// TIA Portal V18 export
// export: Created 2025-12-01T17:52:52.7143684Z, ExportSetting None, DisplayName Totally Integrated Automation Portal, DisplayVersion V18 Update 5, DisplayName TIA Portal Openness, DisplayVersion V18 Update 5, DisplayName TIA Portal Teamcenter Gateway, DisplayVersion V18, DisplayName TIA Portal Version Control Interface, DisplayVersion V18, DisplayName STEP 7 Professional, DisplayVersion V18 Update 5, DisplayName STEP 7 Safety, DisplayVersion V18, DisplayName WinCC Professional, DisplayVersion V18 Update 5
Screen "10MainScreen"  1280x800, Number=10, Template=00MainScreen
  on GenerateScreen: SetBit(Tag := NormalON); ResetBit(Tag := NormalOFF); SetTag(Tag := ST_SysDBNum, Value := 1060); SetTag(Tag := PM_CountCycleDBNum, Value := 1061); SetTag(Tag := ST_PMDBNum, Value := 1063)
  ScreenLayer "Layer_0"
    Button "按钮_4" at 383,725 size 128x75  PictureOff=向右箭头_0, StyleItem=BtnNormal20, TextOff="报 警 / Alarm / Poplach"
      RangeAppearanceAnimation "RangeAppearanceAnimation"
        tag ST_AlarmON
        1..1: back #ff0000, fore #d6d3ce, flashing
      on Click: ActivateScreen(Screen name := 300Main, Object number := 0); SetTag(Tag := Sys_VersionManagement_HMIPageID, Value := 300)
    Button "按钮_6"  Authorization=Manage Parameter, PictureOff=向右箭头_0, StyleItem=BtnNormal20, TextOff="参数设定 / Parameter setting / Parameter nastavenie", TextOn="参数设定 / Parameter setting / Parameter nastavenie"
      RangeAppearanceAnimation "RangeAppearanceAnimation"
        tag _unlock[5]
        0..0: back #d6e1e8, fore #c0c0c0
      on Click: ActivateScreen(Screen name := 700 Main, Object number := 0)
    Button "按钮_8" at 511,725 size 128x75  StyleItem=BtnNormal20, TextOff="MES", TextOn="照明灯 / Light / Svetlo"
      on Press: ActivateScreen(Screen name := 900MES, Object number := 0); SetTag(Tag := Sys_VersionManagement_HMIPageID, Value := 900)
    Button "按钮_11" at 256,725 size 128x75  PictureOff=向右箭头_0, StyleItem=BtnNormal20, TextOff="Safety Status", TextOn="Safety Status"
      on Click: ShowPopupScreen(Name of the screen := Pilz, X coordinate := 350, Y coordinate := 150, Display mode := -1, Animation := -1, Animation speed := 1)
    Button "btnMenu5_1" at 128,725 size 128x75  StyleItem=BtnActive20, TextOff="主页面 / Main", TextOn="主页面 / Main"
      on Click: ActivateScreen(Screen name := , Object number := 0); SetTag(Tag := Sys_VersionManagement_HMIPageID, Value := 10)
    Button "按钮_1"  PictureOff=向右箭头_0, StyleItem=BtnNormal20, TextList=蜂鸣器屏蔽, TextOff="蜂鸣器 屏蔽 / Buzzer shield / Bzučiak štít", TextOn="蜂鸣器 屏蔽 / Buzzer shield"
      RangeAppearanceAnimation "RangeAppearanceAnimation"
        tag ST_CommandBuzzerOn
        1..1: back #3366ff, fore #d6d3ce
      on Click: InvertBit(Tag := ST_CommandBuzzerOn)
      ProcessValue := ST_CommandBuzzerOn
    GraphicView "图形视图_1" at 157,95 size 972x584  Picture=图形_44
    Circle "圆_1" at 259,725 size 29x29
      RangeAppearanceAnimation "RangeAppearanceAnimation"
        tag PilzData_Status
        1..1: back #00ff00, fore #181c31
        2..2: back #ff0000, fore #181c31
    TextField "文本域_14" at 227,649 size 17x28  Text="1"
    TextField "文本域_9" at 1132,93 size 118x42  Text="Current Temperature_1 / Text"
    TextField "文本域_10" at 1132,130 size 118x42  Text="Current Temperature_2 / Text"
    TextField "文本域_11" at 1132,177 size 125x23  Text="SetTemperature / Text"
    TextField "文本域_12" at 1133,213 size 117x23  Text="SetSolidifyTime / Text"
    TextField "文本域_13" at 1132,241 size 92x42  Text="Actual SolidifyTime / Text"
    IOField "I/O 域_1"  FormatPattern=s99999, Mode=Output, ShiftDecimalPoint=1
      ProcessValue := ST10_PLC_GetDB_InData_Data_CurrentTemperature_1
    IOField "I/O 域_2"  FormatPattern=s99999, Mode=Output, ShiftDecimalPoint=1
      ProcessValue := ST10_PLC_GetDB_InData_Data_CurrentTemperature_2
    IOField "I/O 域_3"  FormatPattern=s99999, Mode=Output, ShiftDecimalPoint=1
      ProcessValue := ST10_PLC_GetDB_InData_Data_SetTemperature
    IOField "I/O 域_4"  FormatPattern=s99999, Mode=Output, Unit=min
      ProcessValue := ST10_PLC_GetDB_InData_Data_SetSolidifyTime
    IOField "I/O 域_5"  FormatPattern=s99999, Mode=Output, Unit=min
      ProcessValue := ST10_PLC_GetDB_InData_Data_ActualSolidifyTime
    SymbolicIOField "符号 IO 域_5" at 291,96 size 742x36  Mode=Output, TextList=FlowName5, TextOff="0", TextOn="1"
      ProcessValue := "ST_PMStep[5]"
    Rectangle "矩形_1" at 1037,283 size 176x159
    Circle "圆_17" at 1047,321 size 17x17
      RangeAppearanceAnimation "RangeAppearanceAnimation"
        tag ST10_PLC_GetDB_InData_Global_Beat
        0..0: back #d9d9d9, fore #181c31
        1..1: back #00ff00, fore #181c31
    TextField "文本域_1" at 1079,316 size 48x28  Text="Beat / Text"
    Circle "圆_18" at 1047,349 size 17x17
      RangeAppearanceAnimation "RangeAppearanceAnimation"
        tag ST10_PLC_GetDB_InData_Global_Alarm
        0..0: back #d9d9d9, fore #181c31
        1..1: back #ff0000, fore #181c31
    TextField "文本域_3"  Text="Alarm / Text"
    Circle "圆_19" at 1047,378 size 17x17
      RangeAppearanceAnimation "RangeAppearanceAnimation"
        tag ST10_PLC_GetDB_InData_Global_AutoMode
        1..1: back #00ff00, fore #181c31
        0..0: back #d9d9d9, fore #181c31
    TextField "文本域_5" at 1079,372 size 101x28  Text="AutoMode / Text"
    Circle "圆_20" at 1047,407 size 17x17
      RangeAppearanceAnimation "RangeAppearanceAnimation"
        tag ST10_PLC_GetDB_InData_Global_ManualMode
        1..1: back #00ff00, fore #181c31
        0..0: back #d9d9d9, fore #181c31
    TextField "文本域_6" at 1079,401 size 124x28  Text="ManualMode / Text"
    TextField "文本域_2" at 1064,286 size 139x28  Text="固化炉 / SolidifyStatus"
    Rectangle "矩形_2" at 172,95 size 117x37
    TextField "文本域_4" at 196,100 size 82x28  Text="ROBOT1"
    SymbolicIOField "符号 IO 域_1" at 291,136 size 742x36  Mode=Output, TextList=FlowName8, TextOff="0", TextOn="1"
      ProcessValue := "ST_PMStep[8]"
    Rectangle "矩形_3" at 172,135 size 117x37
    TextField "文本域_7" at 196,140 size 82x28  Text="ROBOT2"
    SymbolicIOField "符号 IO 域_2" at 291,176 size 742x36  Mode=Output, TextList=FlowName15, TextOff="0", TextOn="1"
      ProcessValue := "ST_PMStep[15]"
    Rectangle "矩形_4" at 172,175 size 117x37
    TextField "文本域_8" at 196,180 size 82x28  Text="ROBOT3"
    IOField "I/O 域_6" at 290,644 size 107x32  FormatPattern=999, Unit=%
      ProcessValue := KukaRobot1_CtrlDB_iSpeedValue
    TextField "文本域_15" at 158,648 size 131x28  Text="Robot1Speed:"
    IOField "I/O 域_7" at 541,644 size 107x32  FormatPattern=999, Unit=%
      ProcessValue := KukaRobot2_CtrlDB_iSpeedValue
    TextField "文本域_16" at 409,648 size 131x28  Text="Robot2Speed:"
    IOField "I/O 域_8" at 786,644 size 107x32  FormatPattern=999, Unit=%
      ProcessValue := KukaRobot3_CtrlDB_iSpeedValue
    TextField "文本域_17" at 662,648 size 131x28  Text="Robot3Speed:"
    Group "Group"
      Circle "圆_2" at 317,578 size 24x24
      Circle "圆_3" at 322,583 size 15x15
        RangeAppearanceAnimation "RangeAppearanceAnimation"
          tag HMI_ESTOP
          1..1: back #ff0000, fore #181c31, flashing
          0..0: back #ff0000, fore #181c31
    Group "Group_2"
      Circle "圆_6" at 169,418 size 24x24
      Circle "圆_7" at 174,423 size 15x15
        RangeAppearanceAnimation "RangeAppearanceAnimation"
          tag ESTOP_PB1
          1..1: back #ff0000, fore #181c31, flashing
          0..0: back #ff0000, fore #181c31
    Group "Group_3"
      Circle "圆_8" at 317,320 size 24x24
      Circle "圆_9" at 322,325 size 15x15
        RangeAppearanceAnimation "RangeAppearanceAnimation"
          tag ESTOP_PB7
          1..1: back #ff0000, fore #181c31, flashing
          0..0: back #ff0000, fore #181c31
    Group "Group_4"
      Circle "圆_10" at 287,209 size 24x24
      Circle "圆_11" at 292,214 size 15x15
        RangeAppearanceAnimation "RangeAppearanceAnimation"
          tag ESTOP_PB3
          1..1: back #ff0000, fore #181c31, flashing
          0..0: back #ff0000, fore #181c31
    Group "Group_5"
      Circle "圆_12" at 488,316 size 24x24
      Circle "圆_13" at 493,321 size 15x15
        RangeAppearanceAnimation "RangeAppearanceAnimation"
          tag ESTOP_PB8
          1..1: back #ff0000, fore #181c31, flashing
          0..0: back #ff0000, fore #181c31
    Group "Group_6"
      Circle "圆_14" at 659,312 size 24x24
      Circle "圆_15" at 664,317 size 15x15
        RangeAppearanceAnimation "RangeAppearanceAnimation"
          tag ESTOP_PB9
          1..1: back #ff0000, fore #181c31, flashing
          0..0: back #ff0000, fore #181c31
    Group "Group_7"
      Circle "圆_16" at 450,206 size 24x24
      Circle "圆_21" at 455,211 size 15x15
        RangeAppearanceAnimation "RangeAppearanceAnimation"
          tag ESTOP_PB4
          1..1: back #ff0000, fore #181c31, flashing
          0..0: back #ff0000, fore #181c31
    Group "Group_8"
      Circle "圆_22" at 611,204 size 24x24
      Circle "圆_23" at 616,209 size 15x15
        RangeAppearanceAnimation "RangeAppearanceAnimation"
          tag ESTOP_PB5
          1..1: back #ff0000, fore #181c31, flashing
          0..0: back #ff0000, fore #181c31
    Group "Group_9"
      Circle "圆_24" at 772,205 size 24x24
      Circle "圆_25" at 777,210 size 15x15
        RangeAppearanceAnimation "RangeAppearanceAnimation"
          tag ESTOP_PB6
          1..1: back #ff0000, fore #181c31, flashing
          0..0: back #ff0000, fore #181c31
    Group "Group_10"
      Circle "圆_26" at 1009,320 size 24x24
      Circle "圆_27" at 1014,325 size 15x15
        RangeAppearanceAnimation "RangeAppearanceAnimation"
          tag PilzData_85A1_I12
          0..0: back #ff0000, fore #181c31, flashing
          1..1: back #ff0000, fore #181c31
    Group "Group_12"
      Circle "圆_30" at 855,518 size 24x24
      Circle "圆_31" at 860,523 size 15x15
        RangeAppearanceAnimation "RangeAppearanceAnimation"
          tag ESTOP_PB2
          1..1: back #ff0000, fore #181c31, flashing
          0..0: back #ff0000, fore #181c31
    TextField "文本域_18" at 340,577 size 110x28  Text="HMI ESTOP"
    Group "Group_1"
      Circle "圆_4" at 959,212 size 24x24
      Circle "圆_5" at 964,217 size 15x15
        RangeAppearanceAnimation "RangeAppearanceAnimation"
          tag PilzData_85A1_I13
          0..0: back #ff0000, fore #181c31, flashing
          1..1: back #ff0000, fore #181c31
    TextField "Template_Text field_1" at 855,4 size 299x25  Text="Tool scanning code is running"
      RangeAppearanceAnimation "RangeAppearanceAnimation"
        tag ChangeOver_DB_Global_ScanFixtureFlag
        1..1: back #00ff00, fore #31344a, flashing
      SingleBitVisibilityAnimation "VisibilityAnimation"
        tag ChangeOver_DB_Global_ScanFixtureFlag
    Button "按钮_2"  StyleItem=BtnNormal20, TextOff="清料模式 / Empty Mode / Text", TextOn="清料模式 / Clearing Mode / Text"
      RangeAppearanceAnimation "RangeAppearanceAnimation"
        tag AutoProcessControl_Robot_1_ClearPart
        0..0: back #d6e1e8, fore #000000
        1..1: back #00ff00, fore #000000
      on Click: InvertBit(Tag := AutoProcessControl_Robot_1_ClearPart)
    Button "btnMenu7_6" at 767,725 size 128x75  StyleItem=BtnNormal20
    Button "btnMenu7_9" at 1088,519 size 189x38  TextOff="A1_TableFixtureCode", TextOn="A1_TableFixtureCode"
      on Click: ShowPopupScreen(Name of the screen := A1_TableCode, X coordinate := 10, Y coordinate := 150, Display mode := -1, Animation := -1, Animation speed := 1)
    Circle "圆_28"
      RangeAppearanceAnimation "RangeAppearanceAnimation"
        tag AutoProcessData_GlobalData_Table1CodeOKFlag
        1..1: back #00ff00, fore #181c31
        0..0: back #ff0000, fore #181c31
    Button "btnMenu7_7" at 1088,559 size 189x38  TextOff="A2_TableFixtureCode", TextOn="A2_TableFixtureCode"
      on Click: ShowPopupScreen(Name of the screen := A2_TableCode, X coordinate := 10, Y coordinate := 150, Display mode := -1, Animation := -1, Animation speed := 1)
    Circle "圆_29"
      RangeAppearanceAnimation "RangeAppearanceAnimation"
        tag AutoProcessData_GlobalData_Table2CodeOKFlag
        1..1: back #00ff00, fore #181c31
        0..0: back #ff0000, fore #181c31
    Button "btnMenu7_8" at 1088,599 size 189x38  TextOff="Robot1_FixtureCode", TextOn="Robot1_FixtureCode"
      on Click: ShowPopupScreen(Name of the screen := A1_FixtureCode, X coordinate := 10, Y coordinate := 150, Display mode := -1, Animation := -1, Animation speed := 1)
    Circle "圆_32"
      RangeAppearanceAnimation "RangeAppearanceAnimation"
        tag AutoProcessData_GlobalData_Fixture1CodeOKFlag
        1..1: back #00ff00, fore #181c31
        0..0: back #ff0000, fore #181c31
    Button "btnMenu7_10" at 1088,640 size 189x38  TextOff="Robot3_FixtureCode", TextOn="Robot3_FixtureCode"
      on Click: ShowPopupScreen(Name of the screen := A2_FixtureCode, X coordinate := 10, Y coordinate := 150, Display mode := -1, Animation := -1, Animation speed := 1)
    Circle "圆_33"
      RangeAppearanceAnimation "RangeAppearanceAnimation"
        tag AutoProcessData_GlobalData_Fixture2CodeOKFlag
        1..1: back #00ff00, fore #181c31
        0..0: back #ff0000, fore #181c31
    Button "btnMenu7_11" at 919,559 size 164x38  TextOff="Robot1_GripCode", TextOn="Robot1_GripCode"
      on Click: ShowPopupScreen(Name of the screen := Robot_Grip, X coordinate := 10, Y coordinate := 150, Display mode := -1, Animation := -1, Animation speed := 1)
    Circle "圆_34"
      RangeAppearanceAnimation "RangeAppearanceAnimation"
        tag AutoProcessData_GlobalData_Robot1GripperCodeOKFlag
        1..1: back #00ff00, fore #181c31
        0..0: back #ff0000, fore #181c31
    Button "btnMenu7_13" at 919,599 size 164x38  TextOff="Robot2_GripCode", TextOn="Robot2_GripCode"
      on Click: ShowPopupScreen(Name of the screen := Robot_Grip, X coordinate := 10, Y coordinate := 150, Display mode := -1, Animation := -1, Animation speed := 1)
    Circle "圆_35"
      RangeAppearanceAnimation "RangeAppearanceAnimation"
        tag AutoProcessData_GlobalData_Robot2GripperCodeOKFlag
        1..1: back #00ff00, fore #181c31
        0..0: back #ff0000, fore #181c31
    Button "btnMenu7_14" at 919,640 size 164x38  TextOff="Robot3_GripCode", TextOn="Robot3_GripCode"
      on Click: ShowPopupScreen(Name of the screen := Robot_Grip, X coordinate := 10, Y coordinate := 150, Display mode := -1, Animation := -1, Animation speed := 1)
    Circle "圆_36"
      RangeAppearanceAnimation "RangeAppearanceAnimation"
        tag AutoProcessData_GlobalData_Robot3GripperCodeOKFlag
        1..1: back #00ff00, fore #181c31
        0..0: back #ff0000, fore #181c31
    Group "Group_11"
      Button "btnMenu7_12" at 221,233 size 105x64  TextOff="H- 轴上料 / H- ShaftBelt", TextOn="H- 轴上料 / H- ShaftBelt"
        on Click: ActivateScreen(Screen name := 261_Motor_H1, Object number := 0); SetTag(Tag := Sys_VersionManagement_HMIPageID, Value := 261)
      GraphicIOField "图形 I/O 域_1" at 222,234 size 36x33  PictureList=StationStatus
        ProcessValue := StationStatusH
    Group "Group_13"
      Button "btnMenu7_16" at 396,233 size 105x64  TextOff="J- 磁铁上料 / J- MagnetBelt", TextOn="J- 磁铁上料 / J- MagnetBelt"
        on Click: ActivateScreen(Screen name := 271_Motor_J1, Object number := 0); SetTag(Tag := Sys_VersionManagement_HMIPageID, Value := 271)
      GraphicIOField "图形 I/O 域_2" at 397,234 size 36x33  PictureList=StationStatus
        ProcessValue := StationStatusJ
    Group "Group_14"
      Button "btnMenu7_17" at 568,233 size 105x64  TextOff="K-预留 上料//预留 / K- ReserveBelt", TextOn="K-预留 上料//预留 / K- ReserveBelt"
        on Click: ActivateScreen(Screen name := 281_Motor_K1, Object number := 0); SetTag(Tag := Sys_VersionManagement_HMIPageID, Value := 281)
      GraphicIOField "图形 I/O 域_3" at 569,234 size 36x33  PictureList=StationStatus
        ProcessValue := StationStatusK
    Group "Group_15"
      Button "btnMenu7_18" at 737,233 size 105x64  TextOff="L- 空托盘 / L- UnloadBelt", TextOn="L- 空托盘 / L- UnloadBelt"
        on Click: ActivateScreen(Screen name := 291_Motor_L1, Object number := 0); SetTag(Tag := Sys_VersionManagement_HMIPageID, Value := 291)
      GraphicIOField "图形 I/O 域_4" at 738,234 size 36x33  PictureList=StationStatus
        ProcessValue := StationStatusL
    Group "Group_16"
      Button "btnMenu7_19" at 884,289 size 124x33  TextOff="固化炉 / Solidify", TextOn="固化炉 / Solidify"
        on Click: ShowPopupScreen(Name of the screen := CuringOven, X coordinate := 350, Y coordinate := 150, Display mode := -1, Animation := -1, Animation speed := 1)
      GraphicIOField "图形 I/O 域_5" at 885,290 size 36x33  PictureList=StationStatus
        ProcessValue := Status_Solidify_Status
    Group "Group_17"
      Button "btnMenu7_20" at 252,378 size 122x33  TextOff="F-机器人1 / F-Robot1", TextOn="F-机器人1 / F-Robot1"
        on Click: ActivateScreen(Screen name := 251  Robot_1, Object number := 0)
      GraphicIOField "图形 I/O 域_6" at 253,379 size 36x33  PictureList=StationStatus
        ProcessValue := Status_FRobot_1_Status
    Group "Group_18"
      Button "btnMenu7_21" at 470,378 size 127x33  TextOff="F-机器人2 / F-Robot2", TextOn="F-机器人2 / F-Robot2"
        on Click: ActivateScreen(Screen name := 254  Robot_2, Object number := 0)
      GraphicIOField "图形 I/O 域_7" at 471,379 size 37x33  PictureList=StationStatus
        ProcessValue := Status_FRobot_2_Status
    Group "Group_19"
      Button "btnMenu7_22" at 647,378 size 129x33  TextOff="F-机器人3 / F-Robot3", TextOn="F-机器人3 / F-Robot3"
        on Click: ActivateScreen(Screen name := 257  Robot_3, Object number := 0)
      GraphicIOField "图形 I/O 域_8" at 648,379 size 38x33  PictureList=StationStatus
        ProcessValue := Status_FRobot_3_Status
    Group "Group_21"
      Button "btnMenu7_4" at 570,445 size 113x33  TextOff="B-压机2 / B-Press2", TextOn="B-压机2 / B-Press2"
        on Click: ActivateScreen(Screen name := 227 Kistler_375A1, Object number := 0)
      GraphicIOField "图形 I/O 域_13" at 571,445 size 36x33  PictureList=StationStatus
        ProcessValue := Status_B2Press_Status
    Group "Group_22"
      Button "btnMenu7_3" at 470,483 size 103x33  TextOff="C-Glue", TextOn="C-Glue"
        on Click: ActivateScreen(Screen name := 230_Cylinder, Object number := 0)
      GraphicIOField "图形 I/O 域_15" at 471,483 size 38x33  PictureList=StationStatus
        ProcessValue := Status_C_Glue_Status
    Group "Group_23"
      Button "btnMenu7_1" at 304,445 size 113x33  TextOff="B-压机1 / B-Press1", TextOn="B-压机1 / B-Press1"
        on Click: ActivateScreen(Screen name := 221 Kistler__372A1, Object number := 0)
      GraphicIOField "图形 I/O 域_12" at 305,445 size 36x33  PictureList=StationStatus
        ProcessValue := Status_B1Press_Status
    Group "Group_24"
      Button "btnMenu7_24" at 159,445 size 117x33  TextOff="E-NG盒1 / E-NG1", TextOn="E-NG盒1 / E-NG1"
        on Click: ActivateScreen(Screen name := 240_Cylinder_E1, Object number := 0)
      GraphicIOField "图形 I/O 域_11" at 160,445 size 38x33  PictureList=StationStatus
        ProcessValue := Status_ENG_1_Status
    Group "Group_25"
      Button "btnMenu7_2" at 191,497 size 124x46  TextOff="A-Ring1 上料 / A-Load Ring1", TextOn="A-Ring1 上料 / A-Load Ring1"
        on Click: ActivateScreen(Screen name := 210_Cylinder_A1, Object number := 0)
      GraphicIOField "图形 I/O 域_9" at 192,498 size 45x44  PictureList=StationStatus
        ProcessValue := Status_A1TableScanStatus
    Group "Group_20"
      Button "btnMenu7_5" at 735,498 size 117x46  TextOff="A-Ring2 上料 / A-Load Ring2", TextOn="A-Ring2 上料 / A-Load Ring2"
        on Click: ActivateScreen(Screen name := 216_Cylinder_A2, Object number := 0)
      GraphicIOField "图形 I/O 域_14" at 735,497 size 42x46  PictureList=StationStatus
        ProcessValue := Status_A2TableScanStatus
    Group "Group_26"
      Button "btnMenu7_23" at 763,425 size 147x33  TextOff="E-NG盒2 / E-NG2", TextOn="E-NG盒2 / E-NG2"
        on Click: ActivateScreen(Screen name := 246_Cylinder_E2, Object number := 0)
      GraphicIOField "图形 I/O 域_10" at 764,425 size 50x33  PictureList=StationStatus
        ProcessValue := Status_ENG_2_Status
    Button "btnMenu7_15" at 639,725 size 128x75  StyleItem=BtnNormal20, TextOff="Process data Layout", TextOn="Process data Layout"
      on Click: ActivateScreen(Screen name := 130 Process Data Layout, Object number := 0)
